LIN {X 0,Y 79.684,Z 683.219,A -85,B 0,C 180,E1 -28132.538,E2 -28132.538} C_VEL
LIN {X 0,Y 74.271,Z 683.779,A -85,B 0,C 180,E1 -28141.759,E2 -28141.759} C_VEL
LIN {X 0,Y 70.911,Z 683.469,A -85,B 0,C 180,E1 -28152.7,E2 -28152.7} C_VEL
LIN {X 0,Y 70.164,Z 682.087,A -85,B 0,C 180,E1 -28164.249,E2 -28164.249} C_VEL
LIN {X 0,Y 70.567,Z 680.973,A -85,B 0,C 180,E1 -28169.997,E2 -28169.997} C_VEL
LIN {X 0,Y 70.264,Z 679.42,A -85,B 0,C 180,E1 -28175.737,E2 -28175.737} C_VEL
LIN {X 0,Y 71.113,Z 675.284,A -85,B 0,C 180,E1 -28187.243,E2 -28187.243} C_VEL
LIN {X 0,Y 74.399,Z 669.724,A -85,B 0,C 180,E1 -28198.181,E2 -28198.181} C_VEL
LIN {X 0,Y 79.923,Z 662.59,A -85,B 0,C 180,E1 -28207.987,E2 -28207.987} C_VEL
LIN {X 0,Y 86.455,Z 654.955,A -85,B 0,C 180,E1 -28215.336,E2 -28215.336} C_VEL
LIN {X 0,Y 92.93,Z 647.165,A -85,B 0,C 180,E1 -28220.816,E2 -28220.816} C_VEL
LIN {X 0,Y 101.429,Z 636.363,A -85,B 0,C 180,E1 -28226.246,E2 -28226.246} C_VEL
LIN {X 0,Y 105.331,Z 631.06,A -85,B 0,C 180,E1 -28228.283,E2 -28228.283} C_VEL
LIN {X 0,Y 107.707,Z 624.374,A -85,B 0,C 180,E1 -28231.577,E2 -28231.577} C_VEL
LIN {X 0,Y 110.152,Z 615.435,A -85,B 0,C 180,E1 -28235.784,E2 -28235.784} C_VEL
LIN {X 0,Y 110.382,Z 612.346,A -85,B 0,C 180,E1 -28237.543,E2 -28237.543} C_VEL
LIN {X 0,Y 109.9,Z 602.888,A -85,B 0,C 180,E1 -28243.574,E2 -28243.574} C_VEL
LIN {X 0,Y 109.347,Z 596.511,A -85,B 0,C 180,E1 -28247.944,E2 -28247.944} C_VEL
LIN {X 0,Y 108.576,Z 590.687,A -85,B 0,C 180,E1 -28252.563,E2 -28252.563} C_VEL
LIN {X 0,Y 107.444,Z 587.222,A -85,B 0,C 180,E1 -28256.251,E2 -28256.251} C_VEL
LIN {X 0,Y 105.898,Z 583.218,A -85,B 0,C 180,E1 -28261.903,E2 -28261.903} C_VEL
LIN {X 0,Y 104.563,Z 580.151,A -85,B 0,C 180,E1 -28267.727,E2 -28267.727} C_VEL
LIN {X 0,Y 103.638,Z 579.351,A -85,B 0,C 180,E1 -28271.74,E2 -28271.74} C_VEL
LIN {X 0,Y 102.616,Z 578.621,A -85,B 0,C 180,E1 -28280.027,E2 -28280.027} C_VEL
LIN {X 0,Y 102.846,Z 579.347,A -85,B 0,C 180,E1 -28288.579,E2 -28288.579} C_VEL
LIN {X 0,Y 103.403,Z 580.382,A -85,B 0,C 180,E1 -28292.941,E2 -28292.941} C_VEL
LIN {X 0,Y 104.582,Z 583.261,A -85,B 0,C 180,E1 -28299.711,E2 -28299.711} C_VEL
LIN {X 0,Y 106.159,Z 587.907,A -85,B 0,C 180,E1 -28306.74,E2 -28306.74} C_VEL
LIN {X 0,Y 107.817,Z 593.12,A -85,B 0,C 180,E1 -28312.806,E2 -28312.806} C_VEL
LIN {X 0,Y 109.514,Z 599.757,A -85,B 0,C 180,E1 -28319.113,E2 -28319.113} C_VEL
LIN {X 0,Y 110.793,Z 606.301,A -85,B 0,C 180,E1 -28324.505,E2 -28324.505} C_VEL
LIN {X 0,Y 110.621,Z 608.819,A -85,B 0,C 180,E1 -28326.046,E2 -28326.046} C_VEL
LIN {X 0,Y 109.628,Z 611.643,A -85,B 0,C 180,E1 -28327.334,E2 -28327.334} C_VEL
LIN {X 0,Y 107.1,Z 616.164,A -85,B 0,C 180,E1 -28328.9,E2 -28328.9} C_VEL
LIN {X 0,Y 101.044,Z 623.843,A -85,B 0,C 180,E1 -28331.125,E2 -28331.125} C_VEL
LIN {X 0,Y 96.053,Z 629.754,A -85,B 0,C 180,E1 -28333.25,E2 -28333.25} C_VEL
LIN {X 0,Y 87.904,Z 639.633,A -85,B 0,C 180,E1 -28338.473,E2 -28338.473} C_VEL
LIN {X 0,Y 80.279,Z 648.326,A -85,B 0,C 180,E1 -28344.98,E2 -28344.98} C_VEL
LIN {X 0,Y 73.709,Z 655.684,A -85,B 0,C 180,E1 -28352.735,E2 -28352.735} C_VEL
LIN {X 0,Y 68.433,Z 661.839,A -85,B 0,C 180,E1 -28361.856,E2 -28361.856} C_VEL
LIN {X 0,Y 64.608,Z 666.947,A -85,B 0,C 180,E1 -28372.382,E2 -28372.382} C_VEL
LIN {X 0,Y 62.582,Z 671.121,A -85,B 0,C 180,E1 -28384.163,E2 -28384.163} C_VEL
LIN {X 0,Y 62.922,Z 674.601,A -85,B 0,C 180,E1 -28397.916,E2 -28397.916} C_VEL
LIN {X 0,Y 65.481,Z 676.573,A -85,B 0,C 180,E1 -28409.168,E2 -28409.168} C_VEL
LIN {X 0,Y 68.752,Z 677.502,A -85,B 0,C 180,E1 -28416.932,E2 -28416.932} C_VEL
LIN {X 0,Y 73.116,Z 677.932,A -85,B 0,C 180,E1 -28423.996,E2 -28423.996} C_VEL
LIN {X 0,Y 78.432,Z 677.867,A -85,B 0,C 180,E1 -28430.296,E2 -28430.296} C_VEL
LIN {X 0,Y 84.564,Z 677.322,A -85,B 0,C 180,E1 -28435.81,E2 -28435.81} C_VEL
LIN {X 0,Y 91.37,Z 676.296,A -85,B 0,C 180,E1 -28440.521,E2 -28440.521} C_VEL
LIN {X 0,Y 98.708,Z 674.781,A -85,B 0,C 180,E1 -28444.576,E2 -28444.576} C_VEL
LIN {X 0,Y 109.932,Z 671.657,A -85,B 0,C 180,E1 -28449.434,E2 -28449.434} C_VEL
LIN {X 0,Y 122.954,Z 666.999,A -85,B 0,C 180,E1 -28453.657,E2 -28453.657} C_VEL
LIN {X 0,Y 135.369,Z 661.481,A -85,B 0,C 180,E1 -28456.763,E2 -28456.763} C_VEL
LIN {X 0,Y 138.79,Z 659.792,A -85,B 0,C 180,E1 -28457.686,E2 -28457.686} C_VEL
LIN {X 0,Y 137.125,Z 660.863,A -85,B 0,C 180,E1 -28459.364,E2 -28459.364} C_VEL
LIN {X 0,Y 125.05,Z 667.038,A -85,B 0,C 180,E1 -28461.976,E2 -28461.976} C_VEL
LIN {X 0,Y 112.785,Z 672.296,A -85,B 0,C 180,E1 -28465.37,E2 -28465.37} C_VEL
LIN {X 0,Y 98.408,Z 677.39,A -85,B 0,C 180,E1 -28471.016,E2 -28471.016} C_VEL
LIN {X 0,Y 87.847,Z 680.26,A -85,B 0,C 180,E1 -28476.865,E2 -28476.865} C_VEL
LIN {X 0,Y 78.573,Z 682.208,A -85,B 0,C 180,E1 -28484.308,E2 -28484.308} C_VEL
LIN {X 0,Y 71.005,Z 683.194,A -85,B 0,C 180,E1 -28493.565,E2 -28493.565} C_VEL
LIN {X 0,Y 65.699,Z 683.172,A -85,B 0,C 180,E1 -28504.663,E2 -28504.663} C_VEL
LIN {X 0,Y 63.245,Z 682.212,A -85,B 0,C 180,E1 -28517.156,E2 -28517.156} C_VEL
LIN {X 0,Y 63.506,Z 680.18,A -85,B 0,C 180,E1 -28529.997,E2 -28529.997} C_VEL
LIN {X 0,Y 63.184,Z 678.537,A -85,B 0,C 180,E1 -28536.383,E2 -28536.383} C_VEL
LIN {X 0,Y 64.316,Z 674.219,A -85,B 0,C 180,E1 -28549.133,E2 -28549.133} C_VEL
LIN {X 0,Y 68.159,Z 668.467,A -85,B 0,C 180,E1 -28561.031,E2 -28561.031} C_VEL
LIN {X 0,Y 74.382,Z 661.125,A -85,B 0,C 180,E1 -28571.402,E2 -28571.402} C_VEL
LIN {X 0,Y 81.566,Z 653.269,A -85,B 0,C 180,E1 -28578.927,E2 -28578.927} C_VEL
LIN {X 0,Y 89.778,Z 643.768,A -85,B 0,C 180,E1 -28585.276,E2 -28585.276} C_VEL
LIN {X 0,Y 97.608,Z 634.13,A -85,B 0,C 180,E1 -28589.766,E2 -28589.766} C_VEL
LIN {X 0,Y 100.22,Z 630.515,A -85,B 0,C 180,E1 -28591.225,E2 -28591.225} C_VEL
LIN {X 0,Y 103.427,Z 621.427,A -85,B 0,C 180,E1 -28595.941,E2 -28595.941} C_VEL
LIN {X 0,Y 104.768,Z 616.721,A -85,B 0,C 180,E1 -28598.353,E2 -28598.353} C_VEL
LIN {X 0,Y 104.781,Z 608.492,A -85,B 0,C 180,E1 -28603.961,E2 -28603.961} C_VEL
LIN {X 0,Y 104.607,Z 601.067,A -85,B 0,C 180,E1 -28609.354,E2 -28609.354} C_VEL
LIN {X 0,Y 104.086,Z 595.426,A -85,B 0,C 180,E1 -28614.189,E2 -28614.189} C_VEL
LIN {X 0,Y 103.19,Z 592.169,A -85,B 0,C 180,E1 -28618.05,E2 -28618.05} C_VEL
LIN {X 0,Y 101.939,Z 588.346,A -85,B 0,C 180,E1 -28623.955,E2 -28623.955} C_VEL
LIN {X 0,Y 101.178,Z 586.435,A -85,B 0,C 180,E1 -28627.987,E2 -28627.987} C_VEL
LIN {X 0,Y 100.322,Z 585.595,A -85,B 0,C 180,E1 -28632.134,E2 -28632.134} C_VEL
LIN {X 0,Y 99.367,Z 584.969,A -85,B 0,C 180,E1 -28640.712,E2 -28640.712} C_VEL
LIN {X 0,Y 99.31,Z 585.237,A -85,B 0,C 180,E1 -28645.128,E2 -28645.128} C_VEL
LIN {X 0,Y 99.985,Z 586.549,A -85,B 0,C 180,E1 -28652.496,E2 -28652.496} C_VEL
LIN {X 0,Y 100.976,Z 589.745,A -85,B 0,C 180,E1 -28660.044,E2 -28660.044} C_VEL
LIN {X 0,Y 102.125,Z 593.926,A -85,B 0,C 180,E1 -28666.518,E2 -28666.518} C_VEL
LIN {X 0,Y 103.365,Z 598.665,A -85,B 0,C 180,E1 -28672.274,E2 -28672.274} C_VEL
LIN {X 0,Y 104.735,Z 605.788,A -85,B 0,C 180,E1 -28679.429,E2 -28679.429} C_VEL
LIN {X 0,Y 105.671,Z 612.643,A -85,B 0,C 180,E1 -28685.359,E2 -28685.359} C_VEL
LIN {X 0,Y 105.86,Z 616.49,A -85,B 0,C 180,E1 -28688.354,E2 -28688.354} C_VEL
LIN {X 0,Y 97.893,Z 627.443,A -85,B 0,C 180,E1 -28692.237,E2 -28692.237} C_VEL
LIN {X 0,Y 96.053,Z 629.754,A -85,B 0,C 180,E1 -28693.25,E2 -28693.25} C_VEL
LIN {X 0,Y 92.431,Z 633.691,A -85,B 0,C 180,E1 -28694.803,E2 -28694.803} C_VEL
LIN {X 0,Y 85.264,Z 639.718,A -85,B 0,C 180,E1 -28696.904,E2 -28696.904} C_VEL
LIN {X 0,Y 78.005,Z 645.337,A -85,B 0,C 180,E1 -28699.562,E2 -28699.562} C_VEL
LIN {X 0,Y 74.365,Z 648.583,A -85,B 0,C 180,E1 -28702.081,E2 -28702.081} C_VEL
LIN {X 0,Y 66.463,Z 656.804,A -85,B 0,C 180,E1 -28711.444,E2 -28711.444} C_VEL
LIN {X 0,Y 60.117,Z 663.806,A -85,B 0,C 180,E1 -28723.525,E2 -28723.525} C_VEL
LIN {X 0,Y 56.77,Z 668.457,A -85,B 0,C 180,E1 -28735.013,E2 -28735.013} C_VEL
LIN {X 0,Y 55.271,Z 672.815,A -85,B 0,C 180,E1 -28750.272,E2 -28750.272} C_VEL
LIN {X 0,Y 56.266,Z 675.13,A -85,B 0,C 180,E1 -28761.349,E2 -28761.349} C_VEL
LIN {X 0,Y 58.812,Z 676.764,A -85,B 0,C 180,E1 -28771.442,E2 -28771.442} C_VEL
LIN {X 0,Y 65.531,Z 678.194,A -85,B 0,C 180,E1 -28784.853,E2 -28784.853} C_VEL
LIN {X 0,Y 73.851,Z 678.402,A -85,B 0,C 180,E1 -28794.537,E2 -28794.537} C_VEL
LIN {X 0,Y 84.422,Z 677.492,A -85,B 0,C 180,E1 -28802.553,E2 -28802.553} C_VEL
LIN {X 0,Y 95.693,Z 675.484,A -85,B 0,C 180,E1 -28808.445,E2 -28808.445} C_VEL
LIN {X 0,Y 108.309,Z 672.259,A -85,B 0,C 180,E1 -28813.26,E2 -28813.26} C_VEL
LIN {X 0,Y 121.261,Z 667.884,A -85,B 0,C 180,E1 -28816.938,E2 -28816.938} C_VEL
LIN {X 0,Y 125.606,Z 666.204,A -85,B 0,C 180,E1 -28817.973,E2 -28817.973} C_VEL
LIN {X 0,Y 125.792,Z 666.15,A -85,B 0,C 180,E1 -28818.232,E2 -28818.232} C_VEL
LIN {X 0,Y 113.047,Z 671.465,A -85,B 0,C 180,E1 -28821.165,E2 -28821.165} C_VEL
LIN {X 0,Y 100.81,Z 675.689,A -85,B 0,C 180,E1 -28824.998,E2 -28824.998} C_VEL
LIN {X 0,Y 89.231,Z 678.946,A -85,B 0,C 180,E1 -28829.956,E2 -28829.956} C_VEL
LIN {X 0,Y 78.57,Z 681.16,A -85,B 0,C 180,E1 -28836.383,E2 -28836.383} C_VEL
LIN {X 0,Y 67.877,Z 682.572,A -85,B 0,C 180,E1 -28846.447,E2 -28846.447} C_VEL
LIN {X 0,Y 62.031,Z 682.819,A -85,B 0,C 180,E1 -28855.491,E2 -28855.491} C_VEL
LIN {X 0,Y 57.427,Z 682.161,A -85,B 0,C 180,E1 -28868.457,E2 -28868.457} C_VEL
LIN {X 0,Y 56.03,Z 680.533,A -85,B 0,C 180,E1 -28882.791,E2 -28882.791} C_VEL
LIN {X 0,Y 56.426,Z 679.318,A -85,B 0,C 180,E1 -28889.996,E2 -28889.996} C_VEL
LIN {X 0,Y 56.465,Z 675.547,A -85,B 0,C 180,E1 -28904.41,E2 -28904.41} C_VEL
LIN {X 0,Y 59.491,Z 670.346,A -85,B 0,C 180,E1 -28918.195,E2 -28918.195} C_VEL
LIN {X 0,Y 65.366,Z 663.64,A -85,B 0,C 180,E1 -28930.168,E2 -28930.168} C_VEL
LIN {X 0,Y 73.544,Z 655.262,A -85,B 0,C 180,E1 -28939.857,E2 -28939.857} C_VEL
LIN {X 0,Y 81.982,Z 646.254,A -85,B 0,C 180,E1 -28946.697,E2 -28946.697} C_VEL
LIN {X 0,Y 90.79,Z 636.165,A -85,B 0,C 180,E1 -28951.853,E2 -28951.853} C_VEL
LIN {X 0,Y 94.812,Z 630.946,A -85,B 0,C 180,E1 -28953.99,E2 -28953.99} C_VEL
LIN {X 0,Y 98.497,Z 621.627,A -85,B 0,C 180,E1 -28959.1,E2 -28959.1} C_VEL
LIN {X 0,Y 99.054,Z 619.999,A -85,B 0,C 180,E1 -28959.963,E2 -28959.963} C_VEL
LIN {X 0,Y 99.549,Z 612.164,A -85,B 0,C 180,E1 -28965.696,E2 -28965.696} C_VEL
LIN {X 0,Y 99.788,Z 606.138,A -85,B 0,C 180,E1 -28970.386,E2 -28970.386} C_VEL
LIN {X 0,Y 99.696,Z 600.934,A -85,B 0,C 180,E1 -28974.946,E2 -28974.946} C_VEL
LIN {X 0,Y 98.888,Z 597.035,A -85,B 0,C 180,E1 -28980.002,E2 -28980.002} C_VEL
LIN {X 0,Y 97.986,Z 594.04,A -85,B 0,C 180,E1 -28985.11,E2 -28985.11} C_VEL
LIN {X 0,Y 97.554,Z 592.575,A -85,B 0,C 180,E1 -28988.286,E2 -28988.286} C_VEL
LIN {X 0,Y 96.752,Z 591.721,A -85,B 0,C 180,E1 -28992.589,E2 -28992.589} C_VEL
LIN {X 0,Y 96.034,Z 591.258,A -85,B 0,C 180,E1 -28997.951,E2 -28997.951} C_VEL
LIN {X 0,Y 95.87,Z 591.219,A -85,B 0,C 180,E1 -29001.504,E2 -29001.504} C_VEL
LIN {X 0,Y 95.95,Z 591.884,A -85,B 0,C 180,E1 -29008.49,E2 -29008.49} C_VEL
LIN {X 0,Y 96.161,Z 592.311,A -85,B 0,C 180,E1 -29010.772,E2 -29010.772} C_VEL
LIN {X 0,Y 96.715,Z 594.392,A -85,B 0,C 180,E1 -29016.938,E2 -29016.938} C_VEL
LIN {X 0,Y 97.389,Z 597.382,A -85,B 0,C 180,E1 -29022.579,E2 -29022.579} C_VEL
LIN {X 0,Y 98.015,Z 600.637,A -85,B 0,C 180,E1 -29027.437,E2 -29027.437} C_VEL
LIN {X 0,Y 98.878,Z 605.396,A -85,B 0,C 180,E1 -29033.236,E2 -29033.236} C_VEL
LIN {X 0,Y 99.567,Z 610.696,A -85,B 0,C 180,E1 -29038.804,E2 -29038.804} C_VEL
LIN {X 0,Y 100.103,Z 617.473,A -85,B 0,C 180,E1 -29045.089,E2 -29045.089} C_VEL
LIN {X 0,Y 99.564,Z 619.068,A -85,B 0,C 180,E1 -29046.056,E2 -29046.056} C_VEL
LIN {X 0,Y 91.325,Z 629.666,A -85,B 0,C 180,E1 -29050.013,E2 -29050.013} C_VEL
LIN {X 0,Y 82.695,Z 639.626,A -85,B 0,C 180,E1 -29055.232,E2 -29055.232} C_VEL
LIN {X 0,Y 74.365,Z 648.583,A -85,B 0,C 180,E1 -29062.081,E2 -29062.081} C_VEL
LIN {X 0,Y 70.815,Z 651.748,A -85,B 0,C 180,E1 -29064.895,E2 -29064.895} C_VEL
LIN {X 0,Y 63.81,Z 656.431,A -85,B 0,C 180,E1 -29069.323,E2 -29069.323} C_VEL
LIN {X 0,Y 57.037,Z 660.734,A -85,B 0,C 180,E1 -29074.919,E2 -29074.919} C_VEL
LIN {X 0,Y 54.068,Z 663.152,A -85,B 0,C 180,E1 -29079.578,E2 -29079.578} C_VEL
LIN {X 0,Y 50.411,Z 667.466,A -85,B 0,C 180,E1 -29090.693,E2 -29090.693} C_VEL
LIN {X 0,Y 48.267,Z 671.673,A -85,B 0,C 180,E1 -29105.626,E2 -29105.626} C_VEL
LIN {X 0,Y 48.471,Z 673.987,A -85,B 0,C 180,E1 -29116.472,E2 -29116.472} C_VEL
LIN {X 0,Y 50.173,Z 675.879,A -85,B 0,C 180,E1 -29127.194,E2 -29127.194} C_VEL
LIN {X 0,Y 53.372,Z 677.336,A -85,B 0,C 180,E1 -29137.192,E2 -29137.192} C_VEL
LIN {X 0,Y 57.957,Z 678.33,A -85,B 0,C 180,E1 -29145.962,E2 -29145.962} C_VEL
LIN {X 0,Y 63.82,Z 678.883,A -85,B 0,C 180,E1 -29153.675,E2 -29153.675} C_VEL
LIN {X 0,Y 70.588,Z 678.896,A -85,B 0,C 180,E1 -29159.998,E2 -29159.998} C_VEL
LIN {X 0,Y 77.933,Z 678.419,A -85,B 0,C 180,E1 -29165.172,E2 -29165.172} C_VEL
LIN {X 0,Y 85.842,Z 677.463,A -85,B 0,C 180,E1 -29169.422,E2 -29169.422} C_VEL
LIN {X 0,Y 94.15,Z 676.022,A -85,B 0,C 180,E1 -29172.939,E2 -29172.939} C_VEL
LIN {X 0,Y 108.645,Z 672.461,A -85,B 0,C 180,E1 -29177.583,E2 -29177.583} C_VEL
LIN {X 0,Y 105.927,Z 673.435,A -85,B 0,C 180,E1 -29178.903,E2 -29178.903} C_VEL
LIN {X 0,Y 91.859,Z 677.484,A -85,B 0,C 180,E1 -29183.347,E2 -29183.347} C_VEL
LIN {X 0,Y 80.072,Z 680.039,A -85,B 0,C 180,E1 -29188.63,E2 -29188.63} C_VEL
LIN {X 0,Y 69.309,Z 681.633,A -85,B 0,C 180,E1 -29195.783,E2 -29195.783} C_VEL
LIN {X 0,Y 60.091,Z 682.275,A -85,B 0,C 180,E1 -29205.43,E2 -29205.43} C_VEL
LIN {X 0,Y 53.111,Z 682.01,A -85,B 0,C 180,E1 -29218.038,E2 -29218.038} C_VEL
LIN {X 0,Y 49.454,Z 680.719,A -85,B 0,C 180,E1 -29233.484,E2 -29233.484} C_VEL
LIN {X 0,Y 49.371,Z 678.406,A -85,B 0,C 180,E1 -29249.996,E2 -29249.996} C_VEL
LIN {X 0,Y 49.612,Z 674.457,A -85,B 0,C 180,E1 -29266.454,E2 -29266.454} C_VEL
LIN {X 0,Y 53.296,Z 669.077,A -85,B 0,C 180,E1 -29281.83,E2 -29281.83} C_VEL
LIN {X 0,Y 60.064,Z 662.151,A -85,B 0,C 180,E1 -29294.585,E2 -29294.585} C_VEL
LIN {X 0,Y 69.131,Z 653.501,A -85,B 0,C 180,E1 -29304.413,E2 -29304.413} C_VEL
LIN {X 0,Y 76.896,Z 645.713,A -85,B 0,C 180,E1 -29310.25,E2 -29310.25} C_VEL
LIN {X 0,Y 86.366,Z 635.401,A -85,B 0,C 180,E1 -29315.421,E2 -29315.421} C_VEL
LIN {X 0,Y 89.441,Z 631.672,A -85,B 0,C 180,E1 -29316.868,E2 -29316.868} C_VEL
LIN {X 0,Y 93.096,Z 623.567,A -85,B 0,C 180,E1 -29321.589,E2 -29321.589} C_VEL
LIN {X 0,Y 93.597,Z 622.02,A -85,B 0,C 180,E1 -29322.523,E2 -29322.523} C_VEL
LIN {X 0,Y 94.432,Z 614.644,A -85,B 0,C 180,E1 -29328.471,E2 -29328.471} C_VEL
LIN {X 0,Y 94.958,Z 608.626,A -85,B 0,C 180,E1 -29333.628,E2 -29333.628} C_VEL
LIN {X 0,Y 95.035,Z 606.422,A -85,B 0,C 180,E1 -29335.761,E2 -29335.761} C_VEL
LIN {X 0,Y 94.755,Z 603.104,A -85,B 0,C 180,E1 -29340.002,E2 -29340.002} C_VEL
LIN {X 0,Y 94.099,Z 600.222,A -85,B 0,C 180,E1 -29344.889,E2 -29344.889} C_VEL
LIN {X 0,Y 93.703,Z 598.554,A -85,B 0,C 180,E1 -29348.629,E2 -29348.629} C_VEL
LIN {X 0,Y 92.946,Z 597.712,A -85,B 0,C 180,E1 -29353.113,E2 -29353.113} C_VEL
LIN {X 0,Y 92.367,Z 597.332,A -85,B 0,C 180,E1 -29357.721,E2 -29357.721} C_VEL
LIN {X 0,Y 92.071,Z 597.431,A -85,B 0,C 180,E1 -29363.661,E2 -29363.661} C_VEL
LIN {X 0,Y 92.121,Z 597.743,A -85,B 0,C 180,E1 -29367.244,E2 -29367.244} C_VEL
LIN {X 0,Y 92.43,Z 599.148,A -85,B 0,C 180,E1 -29373.245,E2 -29373.245} C_VEL
LIN {X 0,Y 92.728,Z 600.602,A -85,B 0,C 180,E1 -29377.327,E2 -29377.327} C_VEL
LIN {X 0,Y 93.123,Z 603.459,A -85,B 0,C 180,E1 -29382.786,E2 -29382.786} C_VEL
LIN {X 0,Y 93.625,Z 607.32,A -85,B 0,C 180,E1 -29388.65,E2 -29388.65} C_VEL
LIN {X 0,Y 94.117,Z 612.751,A -85,B 0,C 180,E1 -29395.229,E2 -29395.229} C_VEL
LIN {X 0,Y 94.335,Z 618.354,A -85,B 0,C 180,E1 -29401.163,E2 -29401.163} C_VEL
LIN {X 0,Y 94.33,Z 619.52,A -85,B 0,C 180,E1 -29402.312,E2 -29402.312} C_VEL
LIN {X 0,Y 93.887,Z 620.954,A -85,B 0,C 180,E1 -29403.315,E2 -29403.315} C_VEL
LIN {X 0,Y 84.496,Z 632.247,A -85,B 0,C 180,E1 -29407.652,E2 -29407.652} C_VEL
LIN {X 0,Y 76.328,Z 641.09,A -85,B 0,C 180,E1 -29412.591,E2 -29412.591} C_VEL
LIN {X 0,Y 67.752,Z 649.679,A -85,B 0,C 180,E1 -29419.544,E2 -29419.544} C_VEL
LIN {X 0,Y 60.267,Z 656.944,A -85,B 0,C 180,E1 -29428.331,E2 -29428.331} C_VEL
LIN {X 0,Y 54.068,Z 663.152,A -85,B 0,C 180,E1 -29439.578,E2 -29439.578} C_VEL
LIN {X 0,Y 51.383,Z 665.44,A -85,B 0,C 180,E1 -29444.73,E2 -29444.73} C_VEL
LIN {X 0,Y 46.027,Z 668.716,A -85,B 0,C 180,E1 -29453.787,E2 -29453.787} C_VEL
LIN {X 0,Y 42.411,Z 671,A -85,B 0,C 180,E1 -29462.585,E2 -29462.585} C_VEL
LIN {X 0,Y 41.138,Z 672.605,A -85,B 0,C 180,E1 -29470.287,E2 -29470.287} C_VEL
LIN {X 0,Y 41.132,Z 673.106,A -85,B 0,C 180,E1 -29472.965,E2 -29472.965} C_VEL
LIN {X 0,Y 43.735,Z 676.134,A -85,B 0,C 180,E1 -29491.174,E2 -29491.174} C_VEL
LIN {X 0,Y 50.403,Z 678.307,A -85,B 0,C 180,E1 -29507.452,E2 -29507.452} C_VEL
LIN {X 0,Y 60.485,Z 679.369,A -85,B 0,C 180,E1 -29519.997,E2 -29519.997} C_VEL
LIN {X 0,Y 70.947,Z 679.262,A -85,B 0,C 180,E1 -29527.847,E2 -29527.847} C_VEL
LIN {X 0,Y 84.447,Z 677.994,A -85,B 0,C 180,E1 -29534.456,E2 -29534.456} C_VEL
LIN {X 0,Y 93.244,Z 676.555,A -85,B 0,C 180,E1 -29537.545,E2 -29537.545} C_VEL
LIN {X 0,Y 89.27,Z 677.543,A -85,B 0,C 180,E1 -29539.134,E2 -29539.134} C_VEL
LIN {X 0,Y 76.899,Z 679.873,A -85,B 0,C 180,E1 -29543.942,E2 -29543.942} C_VEL
LIN {X 0,Y 65.381,Z 681.321,A -85,B 0,C 180,E1 -29550.686,E2 -29550.686} C_VEL
LIN {X 0,Y 55.208,Z 681.789,A -85,B 0,C 180,E1 -29560.195,E2 -29560.195} C_VEL
LIN {X 0,Y 47.199,Z 681.338,A -85,B 0,C 180,E1 -29573.439,E2 -29573.439} C_VEL
LIN {X 0,Y 42.671,Z 679.957,A -85,B 0,C 180,E1 -29590.763,E2 -29590.763} C_VEL
LIN {X 0,Y 42.294,Z 677.468,A -85,B 0,C 180,E1 -29609.995,E2 -29609.995} C_VEL
LIN {X 0,Y 42.814,Z 673.33,A -85,B 0,C 180,E1 -29629.16,E2 -29629.16} C_VEL
LIN {X 0,Y 47.361,Z 667.758,A -85,B 0,C 180,E1 -29646.404,E2 -29646.404} C_VEL
LIN {X 0,Y 55.183,Z 660.61,A -85,B 0,C 180,E1 -29659.824,E2 -29659.824} C_VEL
LIN {X 0,Y 63.883,Z 652.947,A -85,B 0,C 180,E1 -29668.488,E2 -29668.488} C_VEL
LIN {X 0,Y 73.583,Z 643.667,A -85,B 0,C 180,E1 -29675.134,E2 -29675.134} C_VEL
LIN {X 0,Y 82.552,Z 634.289,A -85,B 0,C 180,E1 -29679.459,E2 -29679.459} C_VEL
LIN {X 0,Y 84.159,Z 632.446,A -85,B 0,C 180,E1 -29680.116,E2 -29680.116} C_VEL
LIN {X 0,Y 87.661,Z 625.745,A -85,B 0,C 180,E1 -29684.157,E2 -29684.157} C_VEL
LIN {X 0,Y 88.169,Z 624.394,A -85,B 0,C 180,E1 -29685.107,E2 -29685.107} C_VEL
LIN {X 0,Y 89.578,Z 616.42,A -85,B 0,C 180,E1 -29692.11,E2 -29692.11} C_VEL
LIN {X 0,Y 90.192,Z 611.753,A -85,B 0,C 180,E1 -29696.651,E2 -29696.651} C_VEL
LIN {X 0,Y 90.308,Z 609.054,A -85,B 0,C 180,E1 -29700.002,E2 -29700.002} C_VEL
LIN {X 0,Y 89.945,Z 606.253,A -85,B 0,C 180,E1 -29704.677,E2 -29704.677} C_VEL
LIN {X 0,Y 89.633,Z 604.367,A -85,B 0,C 180,E1 -29709.024,E2 -29709.024} C_VEL
LIN {X 0,Y 88.901,Z 603.573,A -85,B 0,C 180,E1 -29713.721,E2 -29713.721} C_VEL
LIN {X 0,Y 88.365,Z 603.258,A -85,B 0,C 180,E1 -29718.552,E2 -29718.552} C_VEL
LIN {X 0,Y 88.144,Z 603.329,A -85,B 0,C 180,E1 -29723.497,E2 -29723.497} C_VEL
LIN {X 0,Y 88.123,Z 603.938,A -85,B 0,C 180,E1 -29728.692,E2 -29728.692} C_VEL
LIN {X 0,Y 88.318,Z 605.231,A -85,B 0,C 180,E1 -29733.853,E2 -29733.853} C_VEL
LIN {X 0,Y 88.515,Z 607.439,A -85,B 0,C 180,E1 -29739.437,E2 -29739.437} C_VEL
LIN {X 0,Y 88.71,Z 610.898,A -85,B 0,C 180,E1 -29745.484,E2 -29745.484} C_VEL
LIN {X 0,Y 88.798,Z 614.513,A -85,B 0,C 180,E1 -29750.72,E2 -29750.72} C_VEL
LIN {X 0,Y 88.838,Z 619.107,A -85,B 0,C 180,E1 -29756.377,E2 -29756.377} C_VEL
LIN {X 0,Y 88.796,Z 621.456,A -85,B 0,C 180,E1 -29759.042,E2 -29759.042} C_VEL
LIN {X 0,Y 88.431,Z 622.838,A -85,B 0,C 180,E1 -29760.22,E2 -29760.22} C_VEL
LIN {X 0,Y 78.65,Z 633.95,A -85,B 0,C 180,E1 -29764.532,E2 -29764.532} C_VEL
LIN {X 0,Y 68.561,Z 644.085,A -85,B 0,C 180,E1 -29770.544,E2 -29770.544} C_VEL
LIN {X 0,Y 58.932,Z 652.905,A -85,B 0,C 180,E1 -29778.852,E2 -29778.852} C_VEL
LIN {X 0,Y 50.718,Z 660.234,A -85,B 0,C 180,E1 -29790.004,E2 -29790.004} C_VEL
LIN {X 0,Y 44.011,Z 666.868,A -85,B 0,C 180,E1 -29806.627,E2 -29806.627} C_VEL
LIN {X 0,Y 41.394,Z 670.846,A -85,B 0,C 180,E1 -29821.898,E2 -29821.898} C_VEL
LIN {X 0,Y 41.132,Z 673.106,A -85,B 0,C 180,E1 -29832.965,E2 -29832.965} C_VEL
LIN {X 0,Y 41.135,Z 674.527,A -85,B 0,C 180,E1 -29840.937,E2 -29840.937} C_VEL
LIN {X 0,Y 40.929,Z 676.442,A -85,B 0,C 180,E1 -29854.535,E2 -29854.535} C_VEL
LIN {X 0,Y 42.177,Z 677.655,A -85,B 0,C 180,E1 -29865.304,E2 -29865.304} C_VEL
LIN {X 0,Y 44.692,Z 678.434,A -85,B 0,C 180,E1 -29872.349,E2 -29872.349} C_VEL
LIN {X 0,Y 45.885,Z 678.61,A -85,B 0,C 180,E1 -29874.33,E2 -29874.33} C_VEL
LIN {X 0,Y 57.959,Z 679.851,A -85,B 0,C 180,E1 -29886.962,E2 -29886.962} C_VEL
LIN {X 0,Y 72.974,Z 679.614,A -85,B 0,C 180,E1 -29895.611,E2 -29895.611} C_VEL
LIN {X 0,Y 76.665,Z 679.291,A -85,B 0,C 180,E1 -29897.121,E2 -29897.121} C_VEL
LIN {X 0,Y 74.285,Z 679.713,A -85,B 0,C 180,E1 -29898.895,E2 -29898.895} C_VEL
LIN {X 0,Y 62.027,Z 680.94,A -85,B 0,C 180,E1 -29904.975,E2 -29904.975} C_VEL
LIN {X 0,Y 50.873,Z 681.301,A -85,B 0,C 180,E1 -29914.01,E2 -29914.01} C_VEL
LIN {X 0,Y 41.678,Z 680.652,A -85,B 0,C 180,E1 -29927.578,E2 -29927.578} C_VEL
LIN {X 0,Y 36.029,Z 679.111,A -85,B 0,C 180,E1 -29947.032,E2 -29947.032} C_VEL
LIN {X 0,Y 35.226,Z 676.521,A -85,B 0,C 180,E1 -29969.994,E2 -29969.994} C_VEL
LIN {X 0,Y 36.163,Z 672.171,A -85,B 0,C 180,E1 -29992.866,E2 -29992.866} C_VEL
LIN {X 0,Y 41.814,Z 666.374,A -85,B 0,C 180,E1 -30012.238,E2 -30012.238} C_VEL
LIN {X 0,Y 50.852,Z 659.012,A -85,B 0,C 180,E1 -30026.011,E2 -30026.011} C_VEL
LIN {X 0,Y 60.432,Z 651.11,A -85,B 0,C 180,E1 -30034.318,E2 -30034.318} C_VEL
LIN {X 0,Y 70.873,Z 641.585,A -85,B 0,C 180,E1 -30040.387,E2 -30040.387} C_VEL
LIN {X 0,Y 78.72,Z 633.663,A -85,B 0,C 180,E1 -30043.674,E2 -30043.674} C_VEL
LIN {X 0,Y 80.33,Z 631.458,A -85,B 0,C 180,E1 -30044.785,E2 -30044.785} C_VEL
LIN {X 0,Y 82.745,Z 626.969,A -85,B 0,C 180,E1 -30047.743,E2 -30047.743} C_VEL
LIN {X 0,Y 84.436,Z 620.217,A -85,B 0,C 180,E1 -30054.151,E2 -30054.151} C_VEL
LIN {X 0,Y 85.226,Z 616.865,A -85,B 0,C 180,E1 -30057.639,E2 -30057.639} C_VEL
LIN {X 0,Y 85.532,Z 614.89,A -85,B 0,C 180,E1 -30060.002,E2 -30060.002} C_VEL
LIN {X 0,Y 85.496,Z 612.027,A -85,B 0,C 180,E1 -30064.717,E2 -30064.717} C_VEL
LIN {X 0,Y 85.346,Z 610.014,A -85,B 0,C 180,E1 -30069.481,E2 -30069.481} C_VEL
LIN {X 0,Y 84.651,Z 609.257,A -85,B 0,C 180,E1 -30074.424,E2 -30074.424} C_VEL
LIN {X 0,Y 83.993,Z 609.087,A -85,B 0,C 180,E1 -30083.022,E2 -30083.022} C_VEL
LIN {X 0,Y 83.85,Z 610.035,A -85,B 0,C 180,E1 -30090.194,E2 -30090.194} C_VEL
LIN {X 0,Y 83.952,Z 611.636,A -85,B 0,C 180,E1 -30095.876,E2 -30095.876} C_VEL
LIN {X 0,Y 83.883,Z 614.459,A -85,B 0,C 180,E1 -30102.09,E2 -30102.09} C_VEL
LIN {X 0,Y 83.686,Z 618.817,A -85,B 0,C 180,E1 -30109.1,E2 -30109.1} C_VEL
LIN {X 0,Y 83.36,Z 623.43,A -85,B 0,C 180,E1 -30115.317,E2 -30115.317} C_VEL
LIN {X 0,Y 83.245,Z 624.535,A -85,B 0,C 180,E1 -30116.721,E2 -30116.721} C_VEL
LIN {X 0,Y 72.677,Z 635.833,A -85,B 0,C 180,E1 -30121.089,E2 -30121.089} C_VEL
LIN {X 0,Y 62.513,Z 645.368,A -85,B 0,C 180,E1 -30126.832,E2 -30126.832} C_VEL
LIN {X 0,Y 53.035,Z 653.45,A -85,B 0,C 180,E1 -30134.635,E2 -30134.635} C_VEL
LIN {X 0,Y 44.677,Z 660.264,A -85,B 0,C 180,E1 -30145.493,E2 -30145.493} C_VEL
LIN {X 0,Y 38.074,Z 665.977,A -85,B 0,C 180,E1 -30160.642,E2 -30160.642} C_VEL
LIN {X 0,Y 34.536,Z 670.367,A -85,B 0,C 180,E1 -30178.849,E2 -30178.849} C_VEL
LIN {X 0,Y 34.901,Z 674.558,A -85,B 0,C 180,E1 -30203.665,E2 -30203.665} C_VEL
LIN {X 0,Y 38.172,Z 676.611,A -85,B 0,C 180,E1 -30218.389,E2 -30218.389} C_VEL
LIN {X 0,Y 45.885,Z 678.61,A -85,B 0,C 180,E1 -30234.33,E2 -30234.33} C_VEL
LIN {X 0,Y 48.024,Z 679.076,A -85,B 0,C 180,E1 -30238.397,E2 -30238.397} C_VEL
LIN {X 0,Y 53.914,Z 680.185,A -85,B 0,C 180,E1 -30252.061,E2 -30252.061} C_VEL
LIN {X 0,Y 56.925,Z 680.348,A -85,B 0,C 180,E1 -30254.763,E2 -30254.763} C_VEL
LIN {X 0,Y 60.464,Z 680.402,A -85,B 0,C 180,E1 -30256.675,E2 -30256.675} C_VEL
LIN {X 0,Y 59.36,Z 680.564,A -85,B 0,C 180,E1 -30258.699,E2 -30258.699} C_VEL
LIN {X 0,Y 47.232,Z 680.713,A -85,B 0,C 180,E1 -30266.768,E2 -30266.768} C_VEL
LIN {X 0,Y 36.72,Z 679.968,A -85,B 0,C 180,E1 -30280.034,E2 -30280.034} C_VEL
LIN {X 0,Y 29.614,Z 678.225,A -85,B 0,C 180,E1 -30301.657,E2 -30301.657} C_VEL
LIN {X 0,Y 28.149,Z 675.496,A -85,B 0,C 180,E1 -30329.993,E2 -30329.993} C_VEL
LIN {X 0,Y 29.715,Z 670.989,A -85,B 0,C 180,E1 -30358.223,E2 -30358.223} C_VEL
LIN {X 0,Y 36.827,Z 664.982,A -85,B 0,C 180,E1 -30379.75,E2 -30379.75} C_VEL
LIN {X 0,Y 47.22,Z 657.368,A -85,B 0,C 180,E1 -30393.243,E2 -30393.243} C_VEL
LIN {X 0,Y 57.692,Z 649.236,A -85,B 0,C 180,E1 -30400.737,E2 -30400.737} C_VEL
LIN {X 0,Y 68.798,Z 639.412,A -85,B 0,C 180,E1 -30406.022,E2 -30406.022} C_VEL
LIN {X 0,Y 75.099,Z 633.133,A -85,B 0,C 180,E1 -30408.285,E2 -30408.285} C_VEL
LIN {X 0,Y 77.14,Z 630.087,A -85,B 0,C 180,E1 -30410.185,E2 -30410.185} C_VEL
LIN {X 0,Y 78.814,Z 625.408,A -85,B 0,C 180,E1 -30414.886,E2 -30414.886} C_VEL
LIN {X 0,Y 80.32,Z 620.738,A -85,B 0,C 180,E1 -30420.002,E2 -30420.002} C_VEL
LIN {X 0,Y 80.683,Z 618.914,A -85,B 0,C 180,E1 -30422.498,E2 -30422.498} C_VEL
LIN {X 0,Y 80.791,Z 617.541,A -85,B 0,C 180,E1 -30424.992,E2 -30424.992} C_VEL
LIN {X 0,Y 80.848,Z 615.488,A -85,B 0,C 180,E1 -30430.014,E2 -30430.014} C_VEL
LIN {X 0,Y 80.148,Z 614.811,A -85,B 0,C 180,E1 -30435.313,E2 -30435.313} C_VEL
LIN {X 0,Y 79.7,Z 614.66,A -85,B 0,C 180,E1 -30440.656,E2 -30440.656} C_VEL
LIN {X 0,Y 79.349,Z 615.239,A -85,B 0,C 180,E1 -30447.67,E2 -30447.67} C_VEL
LIN {X 0,Y 79.37,Z 616.005,A -85,B 0,C 180,E1 -30452.095,E2 -30452.095} C_VEL
LIN {X 0,Y 79.122,Z 618.275,A -85,B 0,C 180,E1 -30458.449,E2 -30458.449} C_VEL
LIN {X 0,Y 79.003,Z 619.442,A -85,B 0,C 180,E1 -30461.077,E2 -30461.077} C_VEL
LIN {X 0,Y 78.641,Z 621.957,A -85,B 0,C 180,E1 -30465.642,E2 -30465.642} C_VEL
LIN {X 0,Y 78.182,Z 625.348,A -85,B 0,C 180,E1 -30471.009,E2 -30471.009} C_VEL
LIN {X 0,Y 78,Z 626.403,A -85,B 0,C 180,E1 -30472.545,E2 -30472.545} C_VEL
LIN {X 0,Y 76.572,Z 628.182,A -85,B 0,C 180,E1 -30473.378,E2 -30473.378} C_VEL
LIN {X 0,Y 65.587,Z 639.006,A -85,B 0,C 180,E1 -30477.608,E2 -30477.608} C_VEL
LIN {X 0,Y 54.997,Z 648.112,A -85,B 0,C 180,E1 -30483.454,E2 -30483.454} C_VEL
LIN {X 0,Y 44.115,Z 656.519,A -85,B 0,C 180,E1 -30492.928,E2 -30492.928} C_VEL
LIN {X 0,Y 35.206,Z 663.065,A -85,B 0,C 180,E1 -30506.556,E2 -30506.556} C_VEL
LIN {X 0,Y 29.17,Z 668.127,A -85,B 0,C 180,E1 -30525.458,E2 -30525.458} C_VEL
LIN {X 0,Y 26.886,Z 671.946,A -85,B 0,C 180,E1 -30548.345,E2 -30548.345} C_VEL
LIN {X 0,Y 30.243,Z 675.859,A -85,B 0,C 180,E1 -30578.38,E2 -30578.38} C_VEL
LIN {X 0,Y 40.759,Z 678.788,A -85,B 0,C 180,E1 -30600.803,E2 -30600.803} C_VEL
LIN {X 0,Y 49.974,Z 679.968,A -85,B 0,C 180,E1 -30610.107,E2 -30610.107} C_VEL
LIN {X 0,Y 56.925,Z 680.348,A -85,B 0,C 180,E1 -30614.763,E2 -30614.763} C_VEL
LIN {X 0,Y 55.518,Z 680.374,A -85,B 0,C 180,E1 -30615.307,E2 -30615.307} C_VEL
LIN {X 0,Y 50.156,Z 680.238,A -85,B 0,C 180,E1 -30614.529,E2 -30614.529} C_VEL
LIN {X 0,Y 37.679,Z 679.049,A -85,B 0,C 180,E1 -30608.47,E2 -30608.47} C_VEL
LIN {X 0,Y 32.601,Z 678.218,A -85,B 0,C 180,E1 -30603.763,E2 -30603.763} C_VEL
LIN {X 0,Y 28.129,Z 677.12,A -85,B 0,C 180,E1 -30596.803,E2 -30596.803} C_VEL
LIN {X 0,Y 20.752,Z 673.791,A -85,B 0,C 180,E1 -30567.867,E2 -30567.867} C_VEL
LIN {X 0,Y 20.992,Z 669.488,A -85,B 0,C 180,E1 -30529.57,E2 -30529.57} C_VEL
LIN {X 0,Y 28.461,Z 663.745,A -85,B 0,C 180,E1 -30501.06,E2 -30501.06} C_VEL
LIN {X 0,Y 38.248,Z 657.335,A -85,B 0,C 180,E1 -30486.755,E2 -30486.755} C_VEL
LIN {X 0,Y 49.851,Z 649.105,A -85,B 0,C 180,E1 -30477.773,E2 -30477.773} C_VEL
LIN {X 0,Y 60.933,Z 640.167,A -85,B 0,C 180,E1 -30472.487,E2 -30472.487} C_VEL
LIN {X 0,Y 72.073,Z 629.768,A -85,B 0,C 180,E1 -30468.841,E2 -30468.841} C_VEL
LIN {X 0,Y 72.997,Z 628.34,A -85,B 0,C 180,E1 -30467.633,E2 -30467.633} C_VEL
LIN {X 0,Y 73.915,Z 624.539,A -85,B 0,C 180,E1 -30460.484,E2 -30460.484} C_VEL
LIN {X 0,Y 74.397,Z 622.198,A -85,B 0,C 180,E1 -30454.53,E2 -30454.53} C_VEL
LIN {X 0,Y 74.57,Z 621.427,A -85,B 0,C 180,E1 -30451.988,E2 -30451.988} C_VEL
LIN {X 0,Y 74.675,Z 620.722,A -85,B 0,C 180,E1 -30448.074,E2 -30448.074} C_VEL
LIN {X 0,Y 75.106,Z 620.101,A -85,B 0,C 180,E1 -30440.662,E2 -30440.662} C_VEL
LIN {X 0,Y 75.436,Z 620.195,A -85,B 0,C 180,E1 -30436.232,E2 -30436.232} C_VEL
LIN {X 0,Y 76.104,Z 620.779,A -85,B 0,C 180,E1 -30430.645,E2 -30430.645} C_VEL
LIN {X 0,Y 75.85,Z 622.887,A -85,B 0,C 180,E1 -30425.319,E2 -30425.319} C_VEL
LIN {X 0,Y 75.051,Z 625.483,A -85,B 0,C 180,E1 -30421.344,E2 -30421.344} C_VEL
LIN {X 0,Y 73.04,Z 630.264,A -85,B 0,C 180,E1 -30415.864,E2 -30415.864} C_VEL
LIN {X 0,Y 72.033,Z 632.391,A -85,B 0,C 180,E1 -30413.666,E2 -30413.666} C_VEL
LIN {X 0,Y 70.825,Z 633.89,A -85,B 0,C 180,E1 -30412.854,E2 -30412.854} C_VEL
LIN {X 0,Y 59.039,Z 644.542,A -85,B 0,C 180,E1 -30409.112,E2 -30409.112} C_VEL
LIN {X 0,Y 47.625,Z 653.404,A -85,B 0,C 180,E1 -30403.544,E2 -30403.544} C_VEL
LIN {X 0,Y 35.462,Z 661.668,A -85,B 0,C 180,E1 -30393.088,E2 -30393.088} C_VEL
LIN {X 0,Y 25.477,Z 668.271,A -85,B 0,C 180,E1 -30373.589,E2 -30373.589} C_VEL
LIN {X 0,Y 20.847,Z 673.378,A -85,B 0,C 180,E1 -30339.694,E2 -30339.694} C_VEL
LIN {X 0,Y 21.108,Z 674.69,A -85,B 0,C 180,E1 -30327.097,E2 -30327.097} C_VEL
LIN {X 0,Y 23.593,Z 677.34,A -85,B 0,C 180,E1 -30293.423,E2 -30293.423} C_VEL
LIN {X 0,Y 32.59,Z 679.199,A -85,B 0,C 180,E1 -30270.381,E2 -30270.381} C_VEL
LIN {X 0,Y 44.825,Z 680.132,A -85,B 0,C 180,E1 -30258.271,E2 -30258.271} C_VEL
LIN {X 0,Y 43.796,Z 679.93,A -85,B 0,C 180,E1 -30255.657,E2 -30255.657} C_VEL
LIN {X 0,Y 35.501,Z 678.754,A -85,B 0,C 180,E1 -30248.145,E2 -30248.145} C_VEL
LIN {X 0,Y 28.129,Z 677.12,A -85,B 0,C 180,E1 -30236.803,E2 -30236.803} C_VEL
LIN {X 0,Y 23.918,Z 675.89,A -85,B 0,C 180,E1 -30228.141,E2 -30228.141} C_VEL
LIN {X 0,Y 17.118,Z 673.479,A -85,B 0,C 180,E1 -30208.88,E2 -30208.88} C_VEL
LIN {X 0,Y 13.907,Z 671.138,A -85,B 0,C 180,E1 -30182.845,E2 -30182.845} C_VEL
LIN {X 0,Y 14.569,Z 669.117,A -85,B 0,C 180,E1 -30160.202,E2 -30160.202} C_VEL
LIN {X 0,Y 15.45,Z 668.404,A -85,B 0,C 180,E1 -30153.917,E2 -30153.917} C_VEL
LIN {X 0,Y 25.944,Z 662.27,A -85,B 0,C 180,E1 -30126.035,E2 -30126.035} C_VEL
LIN {X 0,Y 37.113,Z 655.536,A -85,B 0,C 180,E1 -30115.39,E2 -30115.39} C_VEL
LIN {X 0,Y 48.583,Z 647.64,A -85,B 0,C 180,E1 -30109.392,E2 -30109.392} C_VEL
LIN {X 0,Y 60.281,Z 638.304,A -85,B 0,C 180,E1 -30105.617,E2 -30105.617} C_VEL
LIN {X 0,Y 67.963,Z 631.25,A -85,B 0,C 180,E1 -30103.631,E2 -30103.631} C_VEL
LIN {X 0,Y 68.932,Z 628.569,A -85,B 0,C 180,E1 -30097.718,E2 -30097.718} C_VEL
LIN {X 0,Y 69.215,Z 627.78,A -85,B 0,C 180,E1 -30095.684,E2 -30095.684} C_VEL
LIN {X 0,Y 69.684,Z 626.321,A -85,B 0,C 180,E1 -30090.286,E2 -30090.286} C_VEL
LIN {X 0,Y 69.999,Z 625.596,A -85,B 0,C 180,E1 -30083.681,E2 -30083.681} C_VEL
LIN {X 0,Y 70.511,Z 625.386,A -85,B 0,C 180,E1 -30077.401,E2 -30077.401} C_VEL
LIN {X 0,Y 71.138,Z 625.875,A -85,B 0,C 180,E1 -30071.398,E2 -30071.398} C_VEL
LIN {X 0,Y 70.72,Z 627.774,A -85,B 0,C 180,E1 -30066.433,E2 -30066.433} C_VEL
LIN {X 0,Y 68.991,Z 631.261,A -85,B 0,C 180,E1 -30061.462,E2 -30061.462} C_VEL
LIN {X 0,Y 67.94,Z 633.282,A -85,B 0,C 180,E1 -30059.02,E2 -30059.02} C_VEL
LIN {X 0,Y 66.802,Z 634.673,A -85,B 0,C 180,E1 -30058.004,E2 -30058.004} C_VEL
LIN {X 0,Y 54.663,Z 645.1,A -85,B 0,C 180,E1 -30055.091,E2 -30055.091} C_VEL
LIN {X 0,Y 42.524,Z 653.917,A -85,B 0,C 180,E1 -30050.491,E2 -30050.491} C_VEL
LIN {X 0,Y 29.67,Z 661.878,A -85,B 0,C 180,E1 -30041.326,E2 -30041.326} C_VEL
LIN {X 0,Y 18.429,Z 668.343,A -85,B 0,C 180,E1 -30019.686,E2 -30019.686} C_VEL
LIN {X 0,Y 13.922,Z 673.301,A -85,B 0,C 180,E1 -29969.985,E2 -29969.985} C_VEL
LIN {X 0,Y 14.816,Z 675.013,A -85,B 0,C 180,E1 -29941.667,E2 -29941.667} C_VEL
LIN {X 0,Y 23.584,Z 677.496,A -85,B 0,C 180,E1 -29906.605,E2 -29906.605} C_VEL
LIN {X 0,Y 29.628,Z 678.391,A -85,B 0,C 180,E1 -29898.392,E2 -29898.392} C_VEL
LIN {X 0,Y 29.278,Z 678.258,A -85,B 0,C 180,E1 -29896.204,E2 -29896.204} C_VEL
LIN {X 0,Y 19.281,Z 675.804,A -85,B 0,C 180,E1 -29879.992,E2 -29879.992} C_VEL
LIN {X 0,Y 13.353,Z 672.92,A -85,B 0,C 180,E1 -29848.227,E2 -29848.227} C_VEL
LIN {X 0,Y 15.45,Z 668.404,A -85,B 0,C 180,E1 -29793.917,E2 -29793.917} C_VEL
LIN {X 0,Y 18.504,Z 666.219,A -85,B 0,C 180,E1 -29778.496,E2 -29778.496} C_VEL
LIN {X 0,Y 24.136,Z 662.179,A -85,B 0,C 180,E1 -29759.228,E2 -29759.228} C_VEL
LIN {X 0,Y 31.086,Z 657.608,A -85,B 0,C 180,E1 -29747.564,E2 -29747.564} C_VEL
LIN {X 0,Y 35.883,Z 654.581,A -85,B 0,C 180,E1 -29744.303,E2 -29744.303} C_VEL
LIN {X 0,Y 48.709,Z 645.915,A -85,B 0,C 180,E1 -29740.763,E2 -29740.763} C_VEL
LIN {X 0,Y 60.775,Z 636.196,A -85,B 0,C 180,E1 -29738.694,E2 -29738.694} C_VEL
LIN {X 0,Y 62.79,Z 634.375,A -85,B 0,C 180,E1 -29738.424,E2 -29738.424} C_VEL
LIN {X 0,Y 63.587,Z 633.269,A -85,B 0,C 180,E1 -29736.687,E2 -29736.687} C_VEL
LIN {X 0,Y 64.14,Z 632.132,A -85,B 0,C 180,E1 -29733.224,E2 -29733.224} C_VEL
LIN {X 0,Y 64.6,Z 631.259,A -85,B 0,C 180,E1 -29729.51,E2 -29729.51} C_VEL
LIN {X 0,Y 64.816,Z 630.81,A -85,B 0,C 180,E1 -29725.706,E2 -29725.706} C_VEL
LIN {X 0,Y 65.299,Z 630.493,A -85,B 0,C 180,E1 -29718.84,E2 -29718.84} C_VEL
LIN {X 0,Y 65.954,Z 630.808,A -85,B 0,C 180,E1 -29712.308,E2 -29712.308} C_VEL
LIN {X 0,Y 65.605,Z 632.127,A -85,B 0,C 180,E1 -29708.394,E2 -29708.394} C_VEL
LIN {X 0,Y 64.714,Z 633.518,A -85,B 0,C 180,E1 -29706.237,E2 -29706.237} C_VEL
LIN {X 0,Y 63.382,Z 635.431,A -85,B 0,C 180,E1 -29703.738,E2 -29703.738} C_VEL
LIN {X 0,Y 50.978,Z 645.673,A -85,B 0,C 180,E1 -29701.955,E2 -29701.955} C_VEL
LIN {X 0,Y 39.551,Z 653.58,A -85,B 0,C 180,E1 -29699.58,E2 -29699.58} C_VEL
LIN {X 0,Y 28.206,Z 660.297,A -85,B 0,C 180,E1 -29695.212,E2 -29695.212} C_VEL
LIN {X 0,Y 14.837,Z 666.98,A -85,B 0,C 180,E1 -29681.277,E2 -29681.277} C_VEL
LIN {X 0,Y 6.842,Z 672.135,A -85,B 0,C 180,E1 -29609.97,E2 -29609.97} C_VEL
LIN {X 0,Y 11.011,Z 674.477,A -85,B 0,C 180,E1 -29550.135,E2 -29550.135} C_VEL
LIN {X 0,Y 14.092,Z 675.155,A -85,B 0,C 180,E1 -29537.57,E2 -29537.57} C_VEL
LIN {X 0,Y 5.607,Z 671.239,A -85,B 0,C 180,E1 -29468.807,E2 -29468.807} C_VEL
LIN {X 0,Y 14.404,Z 666.121,A -85,B 0,C 180,E1 -29400.814,E2 -29400.814} C_VEL
LIN {X 0,Y 25.829,Z 660.363,A -85,B 0,C 180,E1 -29388.937,E2 -29388.937} C_VEL
LIN {X 0,Y 35.883,Z 654.581,A -85,B 0,C 180,E1 -29384.303,E2 -29384.303} C_VEL
LIN {X 0,Y 38.986,Z 652.492,A -85,B 0,C 180,E1 -29382.227,E2 -29382.227} C_VEL
LIN {X 0,Y 43.519,Z 648.995,A -85,B 0,C 180,E1 -29377.278,E2 -29377.278} C_VEL
LIN {X 0,Y 48.185,Z 645.346,A -85,B 0,C 180,E1 -29373.252,E2 -29373.252} C_VEL
LIN {X 0,Y 51.279,Z 642.901,A -85,B 0,C 180,E1 -29372.323,E2 -29372.323} C_VEL
LIN {X 0,Y 58.046,Z 637.39,A -85,B 0,C 180,E1 -29372.064,E2 -29372.064} C_VEL
LIN {X 0,Y 59.379,Z 635.93,A -85,B 0,C 180,E1 -29368.261,E2 -29368.261} C_VEL
LIN {X 0,Y 59.917,Z 635.414,A -85,B 0,C 180,E1 -29360.234,E2 -29360.234} C_VEL
LIN {X 0,Y 60.6,Z 635.535,A -85,B 0,C 180,E1 -29353.415,E2 -29353.415} C_VEL
LIN {X 0,Y 60.326,Z 636.158,A -85,B 0,C 180,E1 -29351.352,E2 -29351.352} C_VEL
LIN {X 0,Y 59.172,Z 637.449,A -85,B 0,C 180,E1 -29350.083,E2 -29350.083} C_VEL
LIN {X 0,Y 46.363,Z 647.448,A -85,B 0,C 180,E1 -29349.864,E2 -29349.864} C_VEL
LIN {X 0,Y 33.869,Z 655.521,A -85,B 0,C 180,E1 -29349.762,E2 -29349.762} C_VEL
LIN {X 0,Y 21.374,Z 662.213,A -85,B 0,C 180,E1 -29349.509,E2 -29349.509} C_VEL
LIN {X 0,Y 7.134,Z 668.365,A -85,B 0,C 180,E1 -29350.078,E2 -29350.078} C_VEL
LIN {X 0,Y 5.974,Z 668.702,A -85,B 0,C 180,E1 -29364.63,E2 -29364.63} C_VEL
LIN {X 0,Y 18.782,Z 663.107,A -85,B 0,C 180,E1 -29372.68,E2 -29372.68} C_VEL
LIN {X 0,Y 33.519,Z 655.128,A -85,B 0,C 180,E1 -29373.011,E2 -29373.011} C_VEL
LIN {X 0,Y 47.87,Z 645.501,A -85,B 0,C 180,E1 -29372.426,E2 -29372.426} C_VEL
LIN {X 0,Y 51.279,Z 642.901,A -85,B 0,C 180,E1 -29372.323,E2 -29372.323} C_VEL
LIN {X 0,Y 51.37,Z 642.773,A -85,B 0,C 180,E1 -29371.451,E2 -29371.451} C_VEL
LIN {X 0,Y 50.199,Z 643.559,A -85,B 0,C 180,E1 -29369.332,E2 -29369.332} C_VEL
LIN {X 0,Y 45.767,Z 646.814,A -85,B 0,C 180,E1 -29364.516,E2 -29364.516} C_VEL
LIN {X 0,Y 40.605,Z 650.516,A -85,B 0,C 180,E1 -29359.775,E2 -29359.775} C_VEL
LIN {X 0,Y 38.348,Z 652.047,A -85,B 0,C 180,E1 -29359.279,E2 -29359.279} C_VEL
LIN {X 0,Y 37.559,Z 652.504,A -85,B 0,C 180,E1 -29360.229,E2 -29360.229} C_VEL
LIN {X 0,Y 37.521,Z 652.517,A -85,B 0,C 180,E1 -29360.541,E2 -29360.541} C_VEL
LIN {X 0,Y 37.561,Z 652.453,A -85,B 0,C 180,E1 -29361.981,E2 -29361.981} C_VEL
LIN {X 0,Y 50.107,Z 643.508,A -85,B 0,C 180,E1 -29364.273,E2 -29364.273} C_VEL
LIN {X 0,Y 54.087,Z 640.327,A -85,B 0,C 180,E1 -29364.566,E2 -29364.566} C_VEL
LIN {X 0,Y 54.649,Z 640.076,A -85,B 0,C 180,E1 -29358.19,E2 -29358.19} C_VEL
LIN {X 0,Y 53.034,Z 641.468,A -85,B 0,C 180,E1 -29357.59,E2 -29357.59} C_VEL
LIN {X 0,Y 40.711,Z 650.444,A -85,B 0,C 180,E1 -29359.728,E2 -29359.728} C_VEL
LIN {X 0,Y 37.521,Z 652.517,A -85,B 0,C 180,E1 -29360.541,E2 -29360.541} C_VEL
LIN {X 0,Y 37.521,Z 652.517,A -85,B 0,C 180,E1 -29360.541,E2 -29360.541}

QRS_NEXT_CUT()

QRS_NEXT()
QRS_HOME()

END
